FUNCTION_BLOCK FB_Axis_NoHoming EXTENDS FB_AxisBase
VAR_INPUT
END_VAR
VAR_OUTPUT
END_VAR
VAR
	fHomePositionSetpoint		: LREAL;
END_VAR

PROPERTY HomePositionSetpoint : LREAL
GET
HomePositionSetpoint := fHomePositionSetpoint;
END_GET
SET
fHomePositionSetpoint := HomePositionSetpoint;
END_SET
END_PROPERTY

METHOD Monitoring : BOOL
VAR_INPUT
END_VAR


SUPER^.Monitoring();		//Called last to allow the bReady bit to be evaluated after all error checking is done
END_METHOD

METHOD MotionControl : BOOL
VAR_INPUT
END_VAR
SUPER^.MotionControl();

fbAxisHome(
			Axis:= SelectedAxis,
			Position:= fHomePositionSetpoint, 
			HomingMode:= MC_Direct,
			bCalibrationCam:= TRUE);
END_METHOD

END_FUNCTION_BLOCK

(* stored: Version 1.1.0.1, ProductVersion 3.1.4024.9
   POU FB_Axis_NoHoming: Id {67f12062-5bd4-44d4-b963-30cd41ea59ee}, SpecialFunc None
   Folder 01_SUPER_Overrides: Id {cfe861f9-eb49-42ec-a7bf-5dfd11116946}
   Property HomePositionSetpoint: Id {f2145d70-a429-4112-b0eb-7f595b2a5dec}
   Get Get: Id {43c4efd8-ef3f-4097-ac83-f65444d8fe77}
   Set Set: Id {4cfd3808-0391-476b-9dfd-8171a5903847}
   Method Monitoring: Id {1c486c59-a8a7-43d8-948e-f34ba8d56c92}
   Method MotionControl: Id {b0ccc3c6-e35f-4a18-adeb-ab31021524ff} *)
